{attribute 'linkalways'} 
{attribute 'no_explicit_call' := 'This FB is a CLASS and must be accessed using methods or properties'}
{attribute 'enable_dynamic_creation'}
FUNCTION_BLOCK FINAL LE_WORD EXTENDS Node
VAR
	in1 : _WORD(0);
	in2 : _WORD(0);
	out : _BOOL(FALSE);
END_VAR

METHOD PUBLIC Clone : I_Node
VAR
	pNode : POINTER TO LE_WORD;
END_VAR
pNode := __NEW(LE_WORD);
Clone := pNode^;
END_METHOD

METHOD FB_init : BOOL
VAR_INPUT
	bInitRetains : BOOL; // if TRUE, the retain variables are initialized (warm start / cold start)
	bInCopyCode : BOOL;  // if TRUE, the instance afterwards gets moved into the copy code (online change)
END_VAR
AddInput('in1',THIS^.in1);
AddInput('in2',THIS^.in2);
AddOutput('out', THIS^.out);
END_METHOD

METHOD PROTECTED OnExecute
VAR
END_VAR
out.Value := in1.Value <= in2.Value;
END_METHOD

END_FUNCTION_BLOCK

(* stored: Version 1.1.0.1, ProductVersion 3.1.4024.15
   POU LE_WORD: Id {a71a9982-48df-4258-a9ce-0592394d2012}, SpecialFunc None
   Folder Constructor: Id {7531b21f-41d8-41b1-bd11-01edefddf296}
   Method Clone: Id {a6919902-6791-4b49-9aed-db05ec59c0a6}
   Method FB_init: Id {f3059397-edab-4d44-a921-a39ded308e7b}
   Method OnExecute: Id {c0ac1eea-d1d9-4557-b884-fc09d7492aa7} *)
